FUNCTION_BLOCK F_MUX_2_2 (* Service Interface Function Block Type *)
  (* Standard: 61499-2 *)
  (* Version 0.0, 2012-05-09, 4DIAC-IDE, 4DIAC-Consortium *)
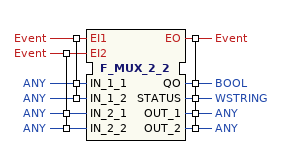
  EVENT_INPUT
    EI1 WITH IN_1_1, IN_1_2; (* event input 1 *)
    EI2 WITH IN_2_1, IN_2_2; (* event input 2 *)
  END_EVENT
  EVENT_OUTPUT
    EO WITH QO, STATUS, OUT_1, OUT_2; (* merge event output *)
  END_EVENT
  VAR_INPUT
    IN_1_1 : ANY;
    IN_1_2 : ANY;
    IN_2_1 : ANY;
    IN_2_2 : ANY;
  END_VAR
  VAR_OUTPUT
    QO : BOOL; (* Event Output Qualifier *)
    STATUS : WSTRING; (* Service Status *)
    OUT_1 : ANY; (* meged data output *)
    OUT_2 : ANY;
  END_VAR
  (* Service APPLICATION/RESOURCE: Service Interface Function Block Type *)
END_FUNCTION_BLOCK
